INTERFACE I_Patlite

PROPERTY bSwitch : BOOL
GET
END_GET
END_PROPERTY

PROPERTY eMachineState : E_MachineState
SET
END_SET
END_PROPERTY

END_INTERFACE

(* stored: Version 1.1.0.1, ProductVersion 3.1.4026.11
   Itf I_Patlite: Id {14c97931-95fa-40c6-b082-3bd22a2a5f82}
   Property bSwitch: Id {9da53c8a-8b53-4b14-8a56-c55a59ce11be}
   Get Get: Id {ca6211ca-c152-4ad4-b15c-1775093ed080}
   Property eMachineState: Id {2c69fe04-fb6b-4907-ad45-1c5badbc4be0}
   Set Set: Id {61f7c06e-b1ad-45a1-8194-7f50bd673af5} *)
